// TIA Portal V17 export
// export: Created 2024-08-07T21:43:51.664276Z, ExportSetting WithDefaults, DisplayName Totally Integrated Automation Portal, DisplayVersion V17 Update 7, DisplayName TIA Portal Openness, DisplayVersion V17 Update 7, DisplayName TIA Portal Version Control Interface, DisplayVersion V17, DisplayName SINAMICS Startdrive Advanced, DisplayVersion V17 SP2, DisplayName SINAMICS Startdrive G110M, G120, G120C, G120D, G120P, G115D, DisplayVersion V17 SP2, DisplayName SINAMICS Startdrive G130, G150, S120, S150, SINAMICS MV, S210, DisplayVersion V17 SP2, DisplayName STEP 7 Professional, DisplayVersion V17 Update 7, DisplayName STEP 7 Safety, DisplayVersion V17 Update 6, DisplayName WinCC Advanced / Unified PC, DisplayVersion V17 Update 7
DATA_BLOCK "AnalogData"   // DB27
{ S7_Optimized_Access := 'FALSE' }
VERSION : 0.1
// stored: AutoNumber false, DBAccessibleFromOPCUA true, DBAccessibleFromWebserver true, IsOnlyStoredInLoadMemory false, IsWriteProtectedInAS false
   VAR
      InputResults : Array[1..12] of Real;
      OutputsRequired : Array[1..8] of Real;
      OutputsRequiredHMI : Array[1..8] of Int;
   END_VAR
BEGIN
   InputResults[1] := 7.960068;
   InputResults[2] := 8.440392;
   InputResults[3] := 7.105035;
   InputResults[4] := 7.011719;
   InputResults[5..12] := 0.0;
   OutputsRequired[1..8] := 0.0;
   OutputsRequiredHMI[1..8] := 16#0000;
END_DATA_BLOCK
